PROGRAM MAIN_ALarm
VAR
	fbAlarmMAIN:						FB_AlarmMAIN;
	fbDiagDataLogging_S:				FB_DiagDataLogging_S;	
	ethercatdiag1,ethercatdiag2:		ethercatinfo_read;
	ec_alarm_trig1,ec_alarm_trig2:		Tc2_Standard.R_TRIG;
	TON_Delay: 							Ton;		
	bInidDone: 							BOOL;
	D1:									DINT:=0;//ec1 报警总数
	D2:									DINT:=0;//ec1报警模块位置
	D3:									DINT:=0;
	D4:									DINT:=0;
    D5,D6:	DINT:=0;
	ModleName1,ModleName2:				Tc2_System.T_MaxString;
	ecnumber1,ecnumber2:				DINT;
	ec_alarm1,ec_alarm2:				BOOL;
	i: 									DINT;

	a,b :INT;
	m1,m2,m3,m4:INT;
	
	Auto_clean_ton:Tc2_Standard.TON;
END_VAR

ethercatdiag_action();

IF NOT bInidDone THEN
	aInit();
ELSE
	TON_Delay(IN:=TRUE , PT:=T#2S );
	IF TON_Delay.Q THEN
		aOtherAlarm();
		fbAlarmMAIN();

		gbAlarm_StopAlarm := fbAlarmMAIN.AlarmAction1;
		gbAlarm_NeedPause := fbAlarmMAIN.AlarmAction2;
		fbDiagDataLogging_s(sInputString:=gsWriteToLog);
		
	END_IF	
END_IF

(*************定时复位历史报警***********************)
Auto_clean_ton(IN:=NOT Auto_clean_ton.Q  , PT:=T#1H , Q=> , ET=> );
IF Auto_clean_ton.Q THEN 
	Alm_bHMIClearHistory:=TRUE;
ELSE 
	Alm_bHMIClearHistory:=FALSE;
END_IF
(*报警灯*)
//GVL_IO.yelllow_lamp:=fbAlarmMAIN.FalshLamp;
(*蜂鸣*)
//GVL_IO.buzz:=fbAlarmMAIN.ShowlampOn;
(*复位*)
//Alm_bBtReset:=GVL_IO.bReast OR gvl.HMI_reset OR GVL.STOM_LBJ.reset;

ACTION aInit:
	AlarmActionArray[1].AlarmMsg.CN	:=	"ETHERCAT 1总线错误,报警数量%D,在第%D个,名称为%S";
	AlarmActionArray[2].AlarmMsg.CN	:=	"ETHERCAT 2总线错误,报警数量%D,在第%D个,名称为%S";


	AlarmActionArray[1].AlarmMsg.EN	:=	'ETHERCAT 1 error,number:%D,deviceID:%D,%S';
	AlarmActionArray[2].AlarmMsg.EN	:=	'ETHERCAT 2 error,number:%D,deviceID:%D,%S';
	AlarmActionArray[3].AlarmMsg.EN	:=	'Alarm3';
	AlarmActionArray[4].AlarmMsg.EN	:=	'Alarm4';
	AlarmActionArray[5].AlarmMsg.EN	:=	'Alarm5';
	AlarmActionArray[6].AlarmMsg.EN	:=	'Alarm6';
	AlarmActionArray[7].AlarmMsg.EN	:=	'Alarm7';
	AlarmActionArray[8].AlarmMsg.EN	:=	'Alarm8';
	AlarmActionArray[9].AlarmMsg.EN	:=	'Alarm9';

	
	
	FOR i:=cnAlarmFirst TO cnAlarmLast DO
		fbSetAlarm[i].EventId := i;
	END_FOR	
	bInidDone:=TRUE;
END_ACTION

ACTION aOtherAlarm:
ec_alarm_trig1(CLK:= ec_alarm1, Q=> );
IF ec_alarm_trig1.Q THEN
	D1:=D1+1;
END_IF
ec_alarm_trig2(CLK:= ec_alarm2, Q=> );
IF ec_alarm_trig2.Q THEN
	D3:=D3+1;
END_IF

fbSetAlarm[1](
	InUse:= TRUE, 
	EventId:= 1, 
	EventActive:= ec_alarm1, 
	QuitRequired:= , 
	QuitEvent:= , 
	EventClass:=Alm_EventClass.Alarm , 
	ToTheLogFile:= TRUE, 
	ToTheHistory:= TRUE, 
	AlarmlampOn:=  TRUE,
	AlarmAction1:= TRUE, 
	AlarmAction2:= TRUE, 
	D1:=			D1,
	D2:=			D2,
	S1:=			ModleName1,
	EventAlive=> , 
	ShowlampOn=> );
	
fbSetAlarm[2](
	InUse:= TRUE, 
	EventId:= 2, 
	EventActive:= ec_alarm2, 
	QuitRequired:= , 
	QuitEvent:= , 
	EventClass:=Alm_EventClass.Alarm ,
	ToTheLogFile:= TRUE, 
	ToTheHistory:= TRUE,
    AlarmlampOn:=  TRUE, 
	AlarmAction1:= TRUE, 
	AlarmAction2:= TRUE, 
	D1:=			D3,
	D2:=			D4,
	S1:=			ModleName2,
	EventAlive=> , 
	ShowlampOn=> );
END_ACTION

ACTION ethercatdiag_action:
ethercatdiag1(
	netID:= , 
	nEcMasterDeviceId:= , 
	slaveAddresses=> , 
	devStates=> , 
	slavenames=> , 
	color=> , 
	nSlaves=> );

IF ethercatdiag1.nSlaves >0 THEN
FOR ecnumber1 :=0 TO (ethercatdiag1.nSlaves-1)  BY 1 DO
	IF ethercatdiag1.devStates[ecnumber1].deviceState>=8 THEN
		ec_alarm1:=FALSE;
	ELSE
		ec_alarm1:=TRUE;
		D2:=ecnumber1+1;
		ModleName1:=ethercatdiag1 .slavenames[ecnumber1];
		EXIT;
	END_IF
END_FOR
END_IF

ethercatdiag2(
	netID:= , 
	nEcMasterDeviceId:= , 
	slaveAddresses=> , 
	devStates=> , 
	slavenames=> , 
	color=> , 
	nSlaves=> );

IF ethercatdiag2.nSlaves >0 THEN
FOR ecnumber2 :=0 TO (ethercatdiag2.nSlaves-1)  BY 1 DO
	IF ethercatdiag2.devStates[ecnumber2].deviceState>=8 THEN
		ec_alarm2:=FALSE;
	ELSE
		ec_alarm2:=TRUE;
		D4:=ecnumber2+1;
		ModleName2:=ethercatdiag2 .slavenames[ecnumber2];
		EXIT;
	END_IF
END_FOR
END_IF
END_ACTION

END_PROGRAM

(* stored: Version 1.1.0.1, ProductVersion 3.1.4024.11
   POU MAIN_Alarm: Id {7b0c7af9-2c6e-4cb2-966d-6fa67d19cf76}, SpecialFunc None
   Action aInit: Id {f2a85357-bf82-43c5-a252-e49c1c204394}
   Action aOtherAlarm: Id {30fcb2e1-b775-4ebc-a6db-5ec0d9869d5c}
   Action ethercatdiag_action: Id {edb01f2c-14ae-442d-97d9-823df92b0ea5} *)
